// TwinCAT 3 PLC project TcoElementsTests
// Title: TcoElementsTests
// Company: Vortex.Library
// ProjectVersion: 0.6.0.913
// ProgramVersion: 3.1.4024.12
// libraries:
//   Tc2_Standard, * (Beckhoff Automation GmbH)
//   Tc2_System, * (Beckhoff Automation GmbH)
//   Tc3_Module, * (Beckhoff Automation GmbH)
//   TcoCore, 0.6.0.913 (Vortex.Library)
//   TcoElements, 0.6.0.913 (Vortex.Library)
//   TcoUtilities, 0.6.0.913 (Vortex.Library)
// project tree:
//   / PlcTask.TcTTO
//   POUs/ MAIN.TcPOU
//   Sandbox/HW_Modules/ AnalogOutputsBase_4.TcDUT, InputsBase_8.TcDUT, AnalogInputsBase_4.TcDUT, OutputsBase_8.TcDUT
//   Sandbox/ IO.TcGVL, TcoElementsSandbox.TcPOU
//   Tests/ TcoDiTests.TcPOU, TcoAiTests.TcPOU, TcoDoTests.TcPOU, TcoAoTests.TcPOU
// (motion and I/O tree: see PLC project tcoelements)
// real-time tasks:
//   TASK PlcTask: cycle T#10ms, priority 20, ADS port 350
//   TASK PlcTask1: cycle T#10ms, priority 21, ADS port 351

CONFIGURATION TcoElementsTests
    RESOURCE PLC ON TwinCAT3
        TASK PlcTask(INTERVAL := T#10ms, PRIORITY := 21);
        PROGRAM MAIN WITH PlcTask : MAIN;
    END_RESOURCE
END_CONFIGURATION

// ---- Sandbox/HW_Modules/AnalogOutputsBase_4.TcDUT
TYPE AnalogOutputsBase_4 :
STRUCT
    {attribute addProperty Name "1"}
    _1 AT %Q* : DINT;
    {attribute addProperty Name "2"}
    _2 AT %Q* : DINT;
    {attribute addProperty Name "3"}
    _3 AT %Q* : DINT;
    {attribute addProperty Name "4"}
    _4 AT %Q* : DINT;
END_STRUCT
END_TYPE

// ---- Sandbox/HW_Modules/InputsBase_8.TcDUT
TYPE InputsBase_8 :
STRUCT
    {attribute addProperty Name "1"}
    _1 AT %I* : BOOL;
    {attribute addProperty Name "2"}
    _2 AT %I* : BOOL;
    {attribute addProperty Name "3"}
    _3 AT %I* : BOOL;
    {attribute addProperty Name "4"}
    _4 AT %I* : BOOL;
    {attribute addProperty Name "5"}
    _5 AT %I* : BOOL;
    {attribute addProperty Name "6"}
    _6 AT %I* : BOOL;
    {attribute addProperty Name "7"}
    _7 AT %I* : BOOL;
    {attribute addProperty Name "8"}
    _8 AT %I* : BOOL;
END_STRUCT
END_TYPE

// ---- Sandbox/HW_Modules/AnalogInputsBase_4.TcDUT
TYPE AnalogInputsBase_4 :
STRUCT
    {attribute addProperty Name "1"}
    _1 AT %I* : INT;
    {attribute addProperty Name "2"}
    _2 AT %I* : DINT;
    {attribute addProperty Name "3"}
    _3 AT %I* : DINT;
    {attribute addProperty Name "4"}
    _4 AT %I* : DINT;
END_STRUCT
END_TYPE

// ---- Sandbox/HW_Modules/OutputsBase_8.TcDUT
TYPE OutputsBase_8 :
STRUCT
    {attribute addProperty Name "1"}
    _1 AT %Q* : BOOL;
    {attribute addProperty Name "2"}
    _2 AT %Q* : BOOL;
    {attribute addProperty Name "3"}
    _3 AT %Q* : BOOL;
    {attribute addProperty Name "4"}
    _4 AT %Q* : BOOL;
    {attribute addProperty Name "5"}
    _5 AT %Q* : BOOL;
    {attribute addProperty Name "6"}
    _6 AT %Q* : BOOL;
    {attribute addProperty Name "7"}
    _7 AT %Q* : BOOL;
    {attribute addProperty Name "8"}
    _8 AT %Q* : BOOL;
END_STRUCT
END_TYPE

// ---- Sandbox/IO.TcGVL
{attribute 'qualified_only'}
{attribute addProperty Name "IO"}
VAR_GLOBAL
    {attribute addProperty Name "A1"}
    A1 : InputsBase_8;
    {attribute addProperty Name "A2"}
    A2 : OutputsBase_8;
    {attribute addProperty Name "A3"}
    A3 : AnalogInputsBase_4;
    {attribute addProperty Name "A4"}
    A4 : AnalogOutputsBase_4;
END_VAR

// ---- POUs/MAIN.TcPOU
PROGRAM MAIN
VAR
    _tcoDigitalSensorTests : TcoDiTests;
    _tcoDigitalActuatorTests : TcoDoTests;
    _tcoAnalogSensorTests : TcoAiTests;
    _tcoAnalogActuatorTests : TcoAoTests;
    _tcoElementsSandbox : TcoElementsSandbox;
END_VAR

_tcoDigitalSensorTests.ProbeRun();
_tcoDigitalActuatorTests.ProbeRun();
_tcoAnalogSensorTests.ProbeRun();
_tcoAnalogActuatorTests.ProbeRun();
_tcoElementsSandbox.Run();

END_PROGRAM

// ---- Tests/TcoDiTests.TcPOU
FUNCTION_BLOCK TcoDiTests EXTENDS TcoCore._internals_TcoContext
VAR
    _signal : BOOL;
    _sut : TcoElements.TcoDi(THIS^);
    _sutNotInitialized : TcoElements.TcoDi(THIS^);
END_VAR
VAR
    _IsTrue_result : BOOL;
    _IsFalse_result : BOOL;
END_VAR

METHOD PROTECTED Main
CASE _testId OF
    50:
        _sutNotInitialized.IsTrue;
        _sutNotInitialized.IsFalse;
        _sutNotInitialized.Service();
        _sutNotInitialized.Restore();
    100:
        _sut(inoSignal := _signal);
        _IsTrue_result := _sut.IsTrue;
    200:
        _sut(inoSignal := _signal);
        _IsFalse_result := _sut.IsFalse;
END_CASE
END_METHOD

END_FUNCTION_BLOCK

// ---- Tests/TcoDoTests.TcPOU
FUNCTION_BLOCK TcoDoTests EXTENDS TcoCore._internals_TcoContext
VAR
    _signal : BOOL;
    _sut : TcoElements.TcoDo(THIS^);
    _sutNotInitialized : TcoElements.TcoDo(THIS^);
END_VAR
VAR
    _IsTrue_result : BOOL;
    _IsFalse_result : BOOL;
END_VAR

METHOD PROTECTED Main
CASE _testId OF
    50:
        _sutNotInitialized.Reset();
        _sutNotInitialized.Set();
        _sutNotInitialized.IsTrue;
        _sutNotInitialized.IsFalse;
        _sutNotInitialized.Service();
        _sutNotInitialized.Restore();
    100:
        _signal := FALSE;
        _sut.Set();
        _sut(inoSignal := _signal);
    150:
        _IsTrue_result := _sut.IsTrue;
        _IsFalse_result := _sut.IsFalse;
    200:
        _signal := TRUE;
        _sut.Reset();
        _sut(inoSignal := _signal);
    250:
        _IsTrue_result := _sut.IsTrue;
        _IsFalse_result := _sut.IsFalse;
END_CASE
END_METHOD

END_FUNCTION_BLOCK

// ---- Tests/TcoAiTests.TcPOU
FUNCTION_BLOCK TcoAiTests EXTENDS TcoCore._internals_TcoContext
VAR
    _signal : DINT;
    _sut : TcoElements.TcoAi(THIS^);
    _sutNotInitialized : TcoElements.TcoAi(THIS^);
END_VAR
VAR
    _ScaledResult : REAL;
END_VAR

METHOD PROTECTED Main
CASE _testId OF
    50:
        _sutNotInitialized.Service();
        _sutNotInitialized.Restore();
    100:
        _sut(inoSignal := _signal);
        _ScaledResult := _sut.Status.Scaled;
END_CASE
END_METHOD

END_FUNCTION_BLOCK

// ---- Tests/TcoAoTests.TcPOU
FUNCTION_BLOCK TcoAoTests EXTENDS TcoCore._internals_TcoContext
VAR
    _signal : DINT;
    _sut : TcoElements.TcoAo(THIS^);
    _sutNotInitialized : TcoElements.TcoAo(THIS^);
END_VAR
VAR
    _UnscaledResult : DINT;
END_VAR

METHOD PROTECTED Main
CASE _testId OF
    50:
        _sutNotInitialized.Service();
        _sutNotInitialized.Restore();
    100:
        _sut(inoSignal := _signal);
        _UnscaledResult := _signal;
    200:
        _sut(inoSignal := _signal);
        _UnscaledResult := REAL_TO_DINT(_sut.Status.Unscaled);
END_CASE
END_METHOD

END_FUNCTION_BLOCK

// ---- Sandbox/TcoElementsSandbox.TcPOU
FUNCTION_BLOCK TcoElementsSandbox EXTENDS TcoCore.TcoContext
VAR
    {attribute addProperty Name "Digital input"}
    _di : TcoElements.TcoDi(THIS^);
    {attribute addProperty Name "Digital output"}
    _do : TcoElements.TcoDo(THIS^);
    _diSignal : BOOL;
    _doSignal : BOOL;
    {attribute addProperty Name "Analogue input"}
    _ai : TcoElements.TcoAi(THIS^);
    {attribute addProperty Name "Analogue input Any"}
    _aiAnyType : TcoElements.TcoAiAny(THIS^);
    {attribute addProperty Name "Analogue output"}
    _ao : TcoElements.TcoAo(THIS^);
    _aiSignal : DINT;
    _aoSignal : DINT;
    {attribute addProperty Name "Carousel"}
    _carousel : TcoElements.TcoCarousel(THIS^);
    codedPosition : WORD;
    {attribute addProperty Name "Disable signal 1"}
    _disableSignal1 : BOOL;
    {attribute addProperty Name "Disable signal 2"}
    _disableSignal2 : BOOL;
END_VAR

METHOD PROTECTED Main
VAR
    _signalInfo : TcoCore.TcoSignalInfo;
END_VAR
_di.Service();
_do.Service();
_di(inoSignal := IO.A1._1);
_do(inoSignal := IO.A2._1);
_Ai.Service();
_aiAnyType.Service();
_Ao.Service();
_Ai(inoSignal := IO.A3._2);
_signalInfo.GetSignalInfo(SIZEOF(IO.A3._1), ADR(IO.A3._1));
_aiAnyType(inSignal := IO.A3._1, inSignalInfo := _signalInfo);
_Ao(inoSignal := IO.A4._1);
_ai.Config.RawLow := 0;
_ai.Config.RawHigh := 65536;
_ai.Config.RealLow := 0.0;
_ai.Config.RealHigh := 100.0;
_carousel.Config.ErrorTime := T#10S;
_carousel.Config.InfoTime := T#2S;
_carousel.Config.Direction := eTcoCarouselDirection.Cw;
_carousel.Config.NumberOfPositions := 8;
_carousel.Config.Offset := 1;

_carousel(inoInPosition := IO.A1._1,
    inoInPrecisePosition := IO.A1._2,
    inoEnableTurn := IO.A2._1,
    inoStartTurn := IO.A2._2,
    inSafetyCondition := IO.A2._3,
    inBasePositionNumber := codedPosition);

_carousel.Suspend(inoDisableCondition := _disableSignal1, Invert := FALSE); //this might be signal from Light Curtain (safety is inerupted)
_carousel.Suspend(inoDisableCondition := _disableSignal2, Invert := TRUE);
_carousel.Suspend(inoDisableCondition := _disableSignal2, Invert := TRUE);
_carousel.SuspendExpression(inDisableCondition := _disableSignal2, inMessage := 'SOME BLOCKIKG ACTIVE');
_carousel.Service();
END_METHOD

END_FUNCTION_BLOCK
